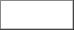
VISUALIZATION VISU_VANNE_2P_V_NoPilot  // 74x30
    Rectangle (0,0 74x30), invisible if: TRUE
    Polygon (50,0)
END_VISUALIZATION

(* stored: Version 1.1.0.1, ProductVersion 3.1.4024.10
   Visu VISU_VANNE_2P_V_NoPilot: Id {a50493c0-2d07-45a9-b20d-768c32b65bee} *)
